FUNCTION_BLOCK _BOOL_TestSuite EXTENDS TcUnit.FB_TestSuite
VAR
END_VAR

TestAddress();
TestClearReference();
TestClone();
TestTypeNameReturnsExpected();
TestMakeReferenceToFollowsReference();
TestMakeReferenceToUpdatesReference();
TestSize();
TestValueReturnsExpectedAfterInit();
TestValueReturnsExpectedAfterChange();
TestSerializeTypeWith();
TestSerializeWith();
TestTryDeserializeFrom();
TestTryMakeReferenceToFollowsReference();
TestTryMakeReferenceToUpdatesReference();

METHOD PUBLIC TestAddress
VAR
    _type : _BOOL(TRUE);
    notExpected : PVOID := 0;
    actual : PVOID;
END_VAR
TEST('TestAddress');

actual := _type.Address;

AssertFalse(
    Condition := (notExpected = actual),
    Message := 'Type did not return a valid address.'
);

TEST_FINISHED();
END_METHOD

METHOD PUBLIC TestClearReference
VAR
    _type : _BOOL(FALSE);
	target : BOOL := FALSE;
    expected : BOOL := FALSE;
    actual : BOOL;
END_VAR
TEST('TestClearReference');

_type.MakeReferenceTo(target);
_type.ClearReference();
target := TRUE;

actual := _type.Value;

AssertEquals(
    Expected := expected,
    Actual := actual,
    Message := 'Value did not follow target change'
);

TEST_FINISHED();
END_METHOD

METHOD PUBLIC TestClone
VAR
    _type : _BOOL(TRUE);
	clone : I_Datatype;
	isValidClone : BOOL;
	compareResult : DINT;
END_VAR
TEST('TestClone');

clone := _type.Clone();

isValidClone := clone <> 0;

IF isValidClone THEN
	compareResult := memcmp(_type.Address, clone.Address, clone.Size);
END_IF

AssertTrue(
	Condition := isValidClone,
	Message := 'Clone did not produce a clone'
);

AssertEquals_DINT(
	Expected := 0,
    Actual := compareResult,
    Message := 'Clone did not return a valid clone.'
);

clone.Dispose();

TEST_FINISHED();
END_METHOD

METHOD PUBLIC TestMakeReferenceToFollowsReference
VAR
    _type : _BOOL(FALSE);
	target : BOOL := FALSE;
    expected : BOOL := TRUE;
    actual : BOOL;
END_VAR
TEST('TestMakeReferenceToFollowsReference');

_type.MakeReferenceTo(target);
target := TRUE;

actual := _type.Value;

AssertEquals(
    Expected := expected,
    Actual := actual,
    Message := 'Value did not follow target change'
);

TEST_FINISHED();
END_METHOD

METHOD PUBLIC TestMakeReferenceToUpdatesReference
VAR
    _type : _BOOL(FALSE);
	target : BOOL := FALSE;
    expected : BOOL := TRUE;
    actual : BOOL;
END_VAR
TEST('TestMakeReferenceToUpdatesReference');

_type.MakeReferenceTo(target);
_type.Value := TRUE;

actual := target;

AssertEquals(
    Expected := expected,
    Actual := actual,
    Message := 'Value did not update target'
);

TEST_FINISHED();
END_METHOD

METHOD PUBLIC TestSerializeTypeWith
VAR
    _type : _BOOL(TRUE);
    serializer : JsonSerializer;
    expected : STRING := '{"typeName":"BOOL"}';
    actual : STRING(500);
END_VAR
TEST('TestSerializeTypeWith');

serializer.Reset();
_type.SerializeTypeWith(serializer);
serializer.TryGetSerializedData(ADR(actual), SIZEOF(actual));

AssertEquals_STRING(
    Expected := expected,
    Actual := actual,
    Message := 'Serialization of type did not return correct string.'
);

TEST_FINISHED();
END_METHOD

METHOD PUBLIC TestSerializeWith
VAR
    _type : _BOOL(TRUE);
    serializer : JsonSerializer;
    expected : STRING := 'true';
    actual : STRING(500);
END_VAR
TEST('TestSerializeWith');

serializer.Reset();
_type.SerializeWith(serializer);
serializer.TryGetSerializedData(ADR(actual), SIZEOF(actual));

AssertEquals_STRING(
    Expected := expected,
    Actual := actual,
    Message := 'Serialization of type data did not return correct string.'
);

TEST_FINISHED();
END_METHOD

METHOD PUBLIC TestSize
VAR
    _type : _BOOL(TRUE);
    expected : UDINT := SIZEOF(BOOL);
    actual : UDINT;
END_VAR
TEST('TestSize');

actual := _type.Size;

AssertEquals_UDINT(
    Expected := Expected,
    Actual := actual,
    Message := 'Type did not return the correct size.'
);

TEST_FINISHED();
END_METHOD

METHOD PUBLIC TestTryDeserializeFrom
VAR
    deserializer : JsonDeserializer;
    feedback : DeserializerFeedback;
    json : STRING := 'true';
    _type : _BOOL(FALSE);
    expected : BOOL := TRUE;
    actual : BOOL;
 END_VAR
TEST('TestTryDeserializeFrom');

deserializer.Reset();
deserializer.TryLoad(json);
_type.TryDeserializeFrom(Deserializer, Feedback);

actual := _type.Value;

AssertEquals(
    Expected := expected,
    Actual := actual,
    Message := 'Type did not deserialize correctly.'
);

TEST_FINISHED();
END_METHOD

METHOD PUBLIC TestTryMakeReferenceToFollowsReference
VAR
    _type : _BOOL(FALSE);
	target : _BOOL(FALSE);
    expected : BOOL := TRUE;
    actual : BOOL;
END_VAR
TEST('TestTryMakeReferenceToFollowsReference');

_type.TryMakeReferenceTo(target);
target.Value := TRUE;

actual := _type.Value;

AssertEquals(
    Expected := expected,
    Actual := actual,
    Message := 'Value did not follow target change'
);

TEST_FINISHED();
END_METHOD

METHOD PUBLIC TestTryMakeReferenceToUpdatesReference
VAR
    _type : _BOOL(FALSE);
	target : _BOOL(FALSE);
    expected : BOOL := TRUE;
    actual : BOOL;
END_VAR
TEST('TestTryMakeReferenceToUpdatesReference');

_type.TryMakeReferenceTo(target);
_type.Value := TRUE;

actual := target.Value;

AssertEquals(
    Expected := expected,
    Actual := actual,
    Message := 'Value did not update target'
);

TEST_FINISHED();
END_METHOD

METHOD PUBLIC TestTypeNameReturnsExpected
VAR
    _type : _BOOL(TRUE);
    expected : STRING := 'BOOL';
    actual : STRING;
END_VAR
TEST('TestTypeNameReturnsExpected');

actual := _type.TypeName;

AssertEquals_STRING(
    Expected := expected,
    Actual := actual,
    Message := 'Type did not return correct iec type.'
);

TEST_FINISHED();
END_METHOD

METHOD PUBLIC TestValueReturnsExpectedAfterChange
VAR
    _type : _BOOL(TRUE);
    expected : BOOL := FALSE;
    actual : BOOL;
END_VAR
TEST('TestValueReturnsExpectedAfterChange');

_type.Value := FALSE;

actual := _type.Value;

AssertEquals(
    Expected := expected,
    Actual := actual,
    Message := 'Expected value not returned after change.'
);

TEST_FINISHED();
END_METHOD

METHOD PUBLIC TestValueReturnsExpectedAfterInit
VAR
    _type : _BOOL(TRUE);
    expected : BOOL := TRUE;
    actual : BOOL;
END_VAR
TEST('TestValueReturnsExpectedAfterInit');

actual := _type.Value;

AssertEquals(
    Expected := expected,
    Actual := actual,
    Message := 'Expected value not returned after Init.'
);

TEST_FINISHED();
END_METHOD

END_FUNCTION_BLOCK

(* stored: Version 1.1.0.1, ProductVersion 3.1.4024.12
   POU _BOOL_TestSuite: Id {392fc7f6-3507-089a-392e-e9b8d35d80dd}, SpecialFunc None
   Method TestAddress: Id {d336854c-b524-45d5-8975-11f5bbf21f62}
   Method TestClearReference: Id {f87e4a0e-2f14-4af3-85f9-5d730459b45d}
   Method TestClone: Id {9773cec8-e870-40e2-b64f-3850df2fca88}
   Method TestMakeReferenceToFollowsReference: Id {57405481-097f-40fd-8e34-f36df45445fd}
   Method TestMakeReferenceToUpdatesReference: Id {a07ef735-752a-46c2-894e-9d1875584159}
   Method TestSerializeTypeWith: Id {ae757e36-0083-4457-bb90-28a58f700ed0}
   Method TestSerializeWith: Id {08058a87-0a98-4e2a-a9b3-e0b3e942ca83}
   Method TestSize: Id {fc668eca-f92a-4308-b792-dc2b6aefbd1a}
   Method TestTryDeserializeFrom: Id {0af62d5f-b7fb-4efc-b8fc-7aa0647249ab}
   Method TestTryMakeReferenceToFollowsReference: Id {923fa26b-da72-4d94-887a-7132568b4bc2}
   Method TestTryMakeReferenceToUpdatesReference: Id {1ccf0b02-3b7b-45b4-9497-7257d3a498ab}
   Method TestTypeNameReturnsExpected: Id {d750e8e3-f129-069b-1a04-7618434ce236}
   Method TestValueReturnsExpectedAfterChange: Id {994c8797-a900-4b60-8992-a5522657990b}
   Method TestValueReturnsExpectedAfterInit: Id {85cbae86-198c-4a25-bfcb-99cb29d1d3dd} *)
